# EPICS StreamDevice protocol: julaboApp/protocol/julaboVariable.proto
#These are the commands where the command string may be different
#for different models of julabo.

#Depending on the julabo model the external temperature
#read command may be "IN_PV_01" or "IN_PV_02".
#So, this uses a parameter from the db file
readExtTemp {
    out "IN_PV_\$1";
    in "%f";
    ExtraInput = Ignore;
}

#Depending on the julabo model the heater power
#read command may be "IN_PV_01" or "IN_PV_02".
#So, this uses a parameter from the db file
readPower {
    out "IN_PV_\$1";
    in "%f";
    ExtraInput = Ignore;
}

#Depending on the julabo model the high limit
#read command may be "IN_SP_01" or "IN_SP_03".
#So, this uses a parameter from the db file
readHighLimit {
    out "IN_SP_\$1";
    in "%f";
    ExtraInput = Ignore;
}

#Depending on the julabo model the high limit
#read command may be "IN_SP_02" or "IN_SP_04".
#So, this uses a parameter from the db file
readLowLimit {
    out "IN_SP_\$1";
    in "%f";
    ExtraInput = Ignore;
}
